// TIA Portal V19 export
TYPE "C501_VAR_IF_BBP_TYPIC"
   STRUCT
      STS_AAN { ExternalAccessible := 'False'; ExternalVisible := 'False'; ExternalWritable := 'False'} : Bool;   // Pomp draait
      BMO_HAND { ExternalAccessible := 'False'; ExternalVisible := 'False'; ExternalWritable := 'False'} : Bool;   // Pomp in hand geschakeld
      TYD_TOT_AAN { ExternalAccessible := 'False'; ExternalVisible := 'False'; ExternalWritable := 'False'} : LInt;   // Totaal aantal draaiuren (in seconden)
      TYD_TOT_AAN_UUR { ExternalAccessible := 'False'; ExternalVisible := 'False'; ExternalWritable := 'False'} : LInt;   // Totaal aantal draaiuren (in uren)
      TYD_AAN { ExternalAccessible := 'False'; ExternalVisible := 'False'; ExternalWritable := 'False'} : Int;   // Aantal seconden dat pomp aangeschakeld is
      TYD_UIT { ExternalAccessible := 'False'; ExternalVisible := 'False'; ExternalWritable := 'False'} : Int;   // Aantal seconden dat pomp uitgeschakeld is
      ENE_MWA1 { ExternalAccessible := 'False'; ExternalVisible := 'False'; ExternalWritable := 'False'} : Real;   // Stroommeting fase 1
      ENE_MWA2 { ExternalAccessible := 'False'; ExternalVisible := 'False'; ExternalWritable := 'False'} : Real;   // Stroommeting fase 2
      ENE_MWA3 { ExternalAccessible := 'False'; ExternalVisible := 'False'; ExternalWritable := 'False'} : Real;   // Stroommeting fase 3
      EXT_HW { ExternalAccessible := 'False'; ExternalVisible := 'False'; ExternalWritable := 'False'} : Bool;   // Sturings hardware (PLC) in storing
      STO { ExternalAccessible := 'False'; ExternalVisible := 'False'; ExternalWritable := 'False'} : Struct   // Opsomming van alle storingen
         A001 : Bool;   // Beveiliging aangesproken
         A002 : Bool;   // Storing van de motorbeveiliging van de pomp
         A003 : Bool;   // Storing softstarter
         A004 : Bool;   // Te hoge temperatuur in de motorwikkelingen
         A005 : Bool;   // De pomp is in onbalans
         A006 : Bool;   // Motorlade uitgeschakeld
         A007 : Bool;   // Motorlade in test
         A008 : Bool;   // Motorlade uitgereden
         A009 : Bool;   // Fout stroommeting fase 1
         A010 : Bool;   // Fout stroommeting fase 2
         A011 : Bool;   // Fout stroommeting fase 3
         A012 : Bool;   // Filter vervuild
         AT01 : Bool;   // Discordantie motor: terugmelding niet ontvangen
         AT02 : Bool;   // Discordantie motor: terugmelding blijft aanwezig
         M001 : Bool;   // Werkschakelaar uitgeschakeld
         M002 : Bool;   // Melding: Pomp heeft te lang niet gedraaid. Periodiek onderhoud nodig
         M003 : Bool;   // Melding: Draaitijd overschrijding
      END_STRUCT;
   END_STRUCT;
END_TYPE
